FUNCTION_BLOCK CoolingNetwork
VAR_INPUT
	//feed temperature setpoint and system enabling
	fSetPointTemperature : REAL;
	bSetStatusOn_eChiller : BOOL;
	bSetStatusOn_HeatPump : BOOL;	
END_VAR
VAR_OUTPUT
	//temperatures in buffer storage
	fTemperatureBufferStorage : REAL;
END_VAR
VAR
	//default parameters
	ST_HVFADefaultParameters : ST_HVFASystemDefaultParameters := (aSetPointLimitsTemperature:=[5,25]);

	//systems
	BufferStorage : FB_BufferStorage;
	eChillerSystem : FB_eChillerSystem;
	HVFAStorage : FB_HVFASystem := (ST_DefaultParameters := ST_HVFADefaultParameters);
	HeatPumpSystem : FB_HeatPumpSystem;
	
	//internal variables
	fAlgorithmPermissionTemperatureRange : REAL := 10; //algorithm mode is only allowed if temperature is between +- 5 K around fSetPointTemperature
	bAlgorithmPermission : BOOL := TRUE;	
END_VAR

//check for algorithm permission
bAlgorithmPermission := Limiter(fInput := BufferStorage.MidTemperature,
								fLowerLimit := fSetPointTemperature-fAlgorithmPermissionTemperatureRange/2,
								fUpperLimit := fSetPointTemperature+fAlgorithmPermissionTemperatureRange);

//buffer storage system
BufferStorage();
fTemperatureBufferStorage := BufferStorage.MidTemperature;

//producer
eChillerSystem(bSetStatusOnAutomatic := bSetStatusOn_eChiller,
	bAlgorithmPermission := bAlgorithmPermission,
	fSetPointAutomatic := fSetPointTemperature,
	fExternalTemperature := BufferStorage.MidTemperature);

//NOTE: heat pump systems contains only two-point actors -> fSetPointAutomatic = 0	
HeatPumpSystem(bSetStatusOnAutomatic := bSetStatusOn_HeatPump,
	bAlgorithmPermission := bAlgorithmPermission,
	fSetPointAutomatic := 0);
	
//external storages

END_FUNCTION_BLOCK

(* stored: Version 1.1.0.1, ProductVersion 3.1.4024.9
   POU CoolingNetwork: Id {155ab526-6067-4e28-9085-03eb63802422}, SpecialFunc None *)
